FUNCTION_BLOCK FB_UpdateSek EXTENDS FB_Basis
VAR_INPUT
	Auswertung		:I_Auswertung;
END_VAR

VAR_OUTPUT
END_VAR

VAR
END_VAR

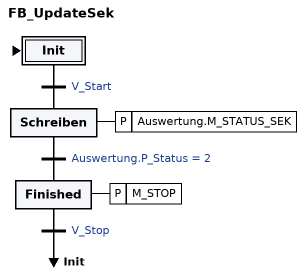
INITIAL_STEP Init:
END_STEP
TRANSITION FROM Init TO Schreiben
    := V_Start;
END_TRANSITION
STEP Schreiben:
    Auswertung.M_STATUS_SEK(P);
END_STEP
TRANSITION FROM Schreiben TO Finished
    := Auswertung.P_Status = 2;
END_TRANSITION
STEP Finished:
    M_STOP(P);
END_STEP
TRANSITION FROM Finished TO Init
    := V_Stop;
END_TRANSITION

END_FUNCTION_BLOCK

(* stored: Version 1.1.0.1, ProductVersion 3.1.4024.12
   POU FB_UpdateSek: Id {433e9bfc-0b7e-4c9f-8881-7127861de752}, SpecialFunc None *)
